// Mitsubishi GX Works2 project: mov한글   PLC: Q02/Q02H

PROGRAM MAIN
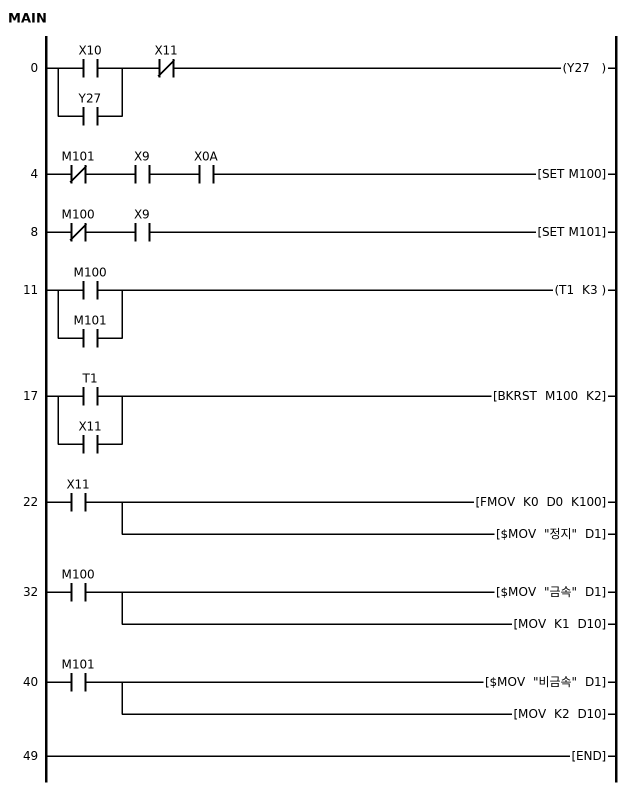
0     LD      X10
      OR      Y27
      ANI     X11
      OUT     Y27
4     LDI     M101
      AND     X9
      AND     X0A
      SET     M100
8     LDI     M100
      AND     X9
      SET     M101
11    LD      M100
      OR      M101
      OUT     T1 K3
17    LD      T1
      OR      X11
      BKRST   M100 K2
22    LD      X11
      FMOV    K0 D0 K100
      $MOV    "정지" D1
32    LD      M100
      $MOV    "금속" D1
      MOV     K1 D10
40    LD      M101
      $MOV    "비금속" D1
      MOV     K2 D10
49    END
END_PROGRAM
